GLOBALCONSTANTS AID_AUXC2 (* Auxiliary control designator type 2 object attribute ids *)
  (* Standard: 61499-1; Description: Copyright (c) 2023 HR Agrartechnik GmbH This program and the accompanying materials are made available under the terms of the Eclipse Public License 2.0 which is available at https://www.eclipse.org/legal/epl-2.0/ SPDX-License-Identifier: EPL-2.0 *)
  (* Version 1.0, 2026-06-20, Franz Höpfinger, HR Agrartechnik GmbH *)
  PACKAGE isobus::UT::Q::const::AID;
  IMPORT eclipse4diac::core::TypeHash;
  VAR_GLOBAL CONSTANT
    PTR_TYPE : USINT := USINT#1; (* 1: AID_AUXC2_PTR_TYPE - Pointer Type: 0=Points to Aux Object, 1=Points to Aux Function/Input assigned to Aux Object, 2=Points to Working Set owner of pointer, 3=Points to Working Set owner of assigned function/input. *)
    OBJ_ID : USINT := USINT#2; (* 2: AID_AUXC2_OBJ_ID - Object ID of a referenced Auxiliary Function or Auxiliary Input object or NULL. *)
  END_VAR
END_GLOBALCONSTANTS
